Fanuc KAREL source: kt00369.KL

-- PROVISIONAL review KL for V940-1; original PC SHA256 e75b428c71dd5999f6ccb0b16fb977cc58881ce7a820bc1e8400254d54f348b4
-- Incomplete behavior may be omitted. Consult companion uncertainty JSON. Do not deploy.
PROGRAM KT00369
%NOLOCKGROUP
VAR
  R1 : REAL
  I2 : INTEGER
  OUT : BOOLEAN
BEGIN
  -- V9_ZERO_TABLE_METADATA_HINT layout=0001; no indexed target words; source/name/runtime held
  -- UNRESOLVED_PC offsets 5-16; opcodes 2E,23
  -- UNRESOLVED_PC offsets 21-32; opcodes 2E,23
  -- UNRESOLVED_PC offsets 37-57; opcodes 21,21,64,70,23
  -- UNRESOLVED_PC offsets 62-66; opcodes 7F
END KT00369
